// TIA Portal V16 export
// export: Created 2021-11-15T20:30:07.621661Z, ExportSetting WithDefaults, DisplayName Totally Integrated Automation Portal, DisplayVersion V16, DisplayName TIA Portal Version Control Interface, DisplayVersion V16, DisplayName TIA Portal Openness, DisplayVersion V16, DisplayName TIA Portal Teamcenter Gateway, DisplayVersion V16, DisplayName STEP 7 Professional, DisplayVersion V16, DisplayName STEP 7 Safety, DisplayVersion V16, DisplayName WinCC Professional, DisplayVersion V16
DATA_BLOCK "Analog scaling output_DB"   // DB3
VERSION : 0.1
// stored: AutoNumber true, InstanceOfName Analog scaling output, InstanceOfType FB
"Analog scaling output"
   // VAR_INPUT
   //    In1 : Bool;
   //    In2 : Bool;
   // END_VAR
   // VAR_OUTPUT
   //    Out20 : Bool;
   // END_VAR
BEGIN
END_DATA_BLOCK
